// TIA Portal V18 export
FUNCTION_BLOCK "lightColumn"   // FB44, FBD
{ S7_Optimized_Access := 'TRUE' }
VERSION : 0.1
// stored: AutoNumber true, IsIECCheckEnabled false, IsRetainMemResEnabled false, MemoryReserve 100, SetENOAutomatically false, UDAEnableTagReadback false
   VAR_INPUT
      er : Bool;
      readyMan : Bool;
      runAuto : Bool;
   END_VAR
   VAR_OUTPUT
      green : Bool;
      red : Bool;
      orange : Bool;
   END_VAR
BEGIN

REGION Network 1
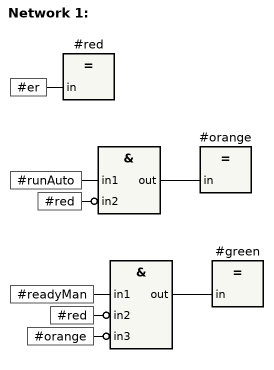
   #red := #er;
   #orange := #runAuto AND NOT #red;
   #green := #readyMan AND NOT #red AND NOT #orange;
END_REGION
END_FUNCTION_BLOCK
